{attribute 'qualified_only'}
VAR_GLOBAL CONSTANT
	FILE_WRITE_BUFFER_SIZE : UDINT := 200000;
END_VAR

(* stored: Version 1.1.0.1, ProductVersion 3.1.4024.4
   GVL GVL_ByteBufferConstants: Id {f290b0e5-6284-42aa-ae06-48716815e922} *)
